FUNCTION_BLOCK Sensor
VAR_INPUT
END_VAR
VAR_OUTPUT
	bSignal  : BOOL;
END_VAR
VAR
	fbSignal : BoolIn;
END_VAR

bSignal := fbSignal.getValue;

PROPERTY getSignal : I_StepCondition
GET
getSignal := fbSignal;
END_GET
END_PROPERTY

END_FUNCTION_BLOCK

(* stored: Version 1.1.0.1, ProductVersion 3.1.4024.2
   POU Sensor: Id {e931cece-00b8-480a-8d07-9e5455c458fa}, SpecialFunc None
   Property getSignal: Id {5a597ac7-fa78-4537-96ce-81a66490c4b6}
   Get Get: Id {6b81593c-a718-48e9-8984-f17bd538bdab} *)
